{attribute 'no_explicit_call' := 'do not call this POU directly'}
FUNCTION_BLOCK INTERNAL FINAL FB_SnappyConfig IMPLEMENTS I_SnappyConfig, I_SnappySetupDefaultsOrRpc, I_SnappySetupConfigSerializer, I_SnappySetupConfigTestFrameWork
VAR
	eConfigState		: (NOT_CONFIGURED, IS_CONFIGURED) := NOT_CONFIGURED;
END_VAR

VAR
	itfSerializerField		: I_Serializer 	:= NULL;
	itfRpcProxyField		: I_RpcProxy	:= NULL;
	itfTestFrameworkField	: I_TestFrameWorkAdapter := NULL;
END_VAR

VAR
	fbJsonSerializer	: FB_JsonSerializer;
	fbRpcProxy			: FB_RpcProxy;
	fbTestNamesProvider : FB_TestSuiteNameProvider;
END_VAR

PROPERTY bIsConfigured : BOOL
GET
bIsConfigured := eConfigState = IS_CONFIGURED;
END_GET
END_PROPERTY

METHOD Build : HRESULT

IF itfRpcProxyField = NULL THEN
	Build := Tc2_System.E_HRESULTAdsErr.INVALIDPARM;
	RETURN;
END_IF

IF itfSerializerField = NULL THEN
	Build := Tc2_System.E_HRESULTAdsErr.INVALIDPARM;
	RETURN;
END_IF

eConfigState := IS_CONFIGURED;
END_METHOD

METHOD Configure : I_SnappySetupDefaultsOrRpc
Configure := THIS^;
IF bIsConfigured THEN
	RETURN;
END_IF
END_METHOD

PROPERTY itfRpcProxy : I_RpcProxy
GET
itfRpcProxy := itfRpcProxyField;
END_GET
END_PROPERTY

PROPERTY itfSerializer : I_Serializer
GET
itfSerializer := itfSerializerField;
END_GET
END_PROPERTY

PROPERTY itfTestFramework : I_TestFrameWorkAdapter
GET
itfTestFramework := itfTestFrameworkField;
END_GET
END_PROPERTY

METHOD UseDefaults : I_SnappySetupConfigTestFrameWork
UseDefaults := THIS^;

IF bIsConfigured THEN
	RETURN;
END_IF

THIS^.itfSerializerField 	:= fbJsonSerializer;
THIS^.itfRpcProxyField 		:= fbRpcProxy;
END_METHOD

METHOD UseRpcProxy : I_SnappySetupConfigSerializer
VAR_INPUT
	itfRpcProxy	: I_RpcProxy;
END_VAR
UseRpcProxy := THIS^;

IF bIsConfigured THEN
	RETURN;
END_IF

THIS^.itfRpcProxyField := itfRpcProxy;
END_METHOD

METHOD UseSerializer : I_SnappySetupConfigBuild
VAR_INPUT
	itfSerializer	: I_Serializer;
END_VAR
UseSerializer := THIS^;

IF bIsConfigured THEN
	RETURN;
END_IF

THIS^.itfSerializerField := itfSerializer;
END_METHOD

METHOD UseTestFramework : I_SnappySetupConfigBuild
VAR_INPUT
	itfTestFramework	: I_TestFrameWorkAdapter;
END_VAR
UseTestFramework := THIS^;

IF bIsConfigured THEN
	RETURN;
END_IF

THIS^.itfTestFrameworkField := itfTestFramework;
END_METHOD

METHOD WithoutTestFramework : I_SnappySetupConfigBuild
VAR_INPUT CONSTANT
	sTestSuiteName 	: T_MaxString;
	sTestName		: T_MaxString;
END_VAR
WithoutTestFramework := THIS^;

THIS^.fbTestNamesProvider.SetTestNames(sTestSuiteName, sTestName);
THIS^.itfTestFrameworkField := THIS^.fbTestNamesProvider;

IF bIsConfigured THEN
	RETURN;
END_IF
END_METHOD

END_FUNCTION_BLOCK

(* stored: Version 1.1.0.1, ProductVersion 3.1.4026.18
   POU FB_SnappyConfig: Id {8454dc2d-fe9a-4b10-b1c8-cd836dfcc8b6}, SpecialFunc None
   Property bIsConfigured: Id {c95bffdc-fb33-45f0-afed-83763b831590}
   Get Get: Id {cb08d6d2-d753-45af-8c4e-f6673ae313d7}
   Method Build: Id {e57235b4-f6fc-486b-ac34-f731fe77b269}
   Method Configure: Id {d4b601e9-973a-4a2e-9dac-fcddd9ce0609}
   Property itfRpcProxy: Id {3acc6c60-e3ab-4391-80f9-91688177f89d}
   Get Get: Id {242c0647-cb67-4957-adba-2ccff583c710}
   Property itfSerializer: Id {246a0fec-3eb1-4c94-8bd4-d64c402ee8ac}
   Get Get: Id {a476cddb-9af0-43ef-aac7-f4aee4a09b21}
   Property itfTestFramework: Id {7daedeaf-667f-4d0a-b8cb-681b5beb3c1d}
   Get Get: Id {2fba5b04-907d-440b-8997-53f107df31bf}
   Method UseDefaults: Id {475c0225-38e9-42f2-aa74-344f1b08102b}
   Method UseRpcProxy: Id {d3dfa10f-48fb-4751-b2fd-3ba4583ad0d8}
   Method UseSerializer: Id {d56172b6-f5cc-4d8d-a7f8-5ecf06e07962}
   Method UseTestFramework: Id {943d3ed1-56e7-4e73-9ea4-64127c6fbebd}
   Method WithoutTestFramework: Id {32f351cd-9643-4f84-95fb-5a9c2326d54d} *)
